Staubli VAL3: RotationTras.dtx

mdesc mNomSpeed
trsf tTransformation = {rx=90}
num nXaxis
num nYaxis
num nZaxis
num nAngle
trsf trNew
num nSetAngle
num nSetXaxis
num nSetYaxis
num nSetZaxis
